(* PLC project Sin nombre, Desconocido Sin nombre 1 *)
(* stored: creationDateTime 2024-04-04T13:22:05, modificationDateTime 2024-04-09T02:45:14 *)

PROGRAM program0
  VAR
    boton_inicio AT %IX0.0 : BOOL;  (* El boton de inicio *)
    boton_parada AT %IX0.1 : BOOL;  (* El boton para detener todo *)
    sensor_caja AT %IW0 : WORD;  (* Entrada con el sensor analogo *)
    motor_cinta AT %QX0.0 : BOOL;  (* Motor para la cinta transportadora *)
    motor_rodillo AT %QX0.1 : BOOL;  (* Motor para activar el rodillo *)
  END_VAR
  VAR
    auxiliar_inicio : BOOL;  (* Variable auxiliar para almacenar si se presiono el boton de inicio *)
    auxiliar_sensor : BOOL;  (* Variable auxiliar para determinar si el sensor esta detectando la caja *)
    auxiliar_reloj : BOOL;  (* Variable auxiliar para determinar si el reloj esta contando *)
    sensor_esta_conectado : BOOL;  (* Comprobacion de que el sensor esta funcionando *)
    sensor_tapado : BOOL;  (* Comprobacion de que el sensor esta siendo tapado *)
  END_VAR
  VAR CONSTANT
    min_luz : WORD := 3500;  (* Minimo de luz requerida para saber si el sensor esta siendo tapado o no *)
    max_tiempo_rodillo : TIME := T#500ms;  (* Maxima cantidad de tiempo por la que el motor del rodillo esta activo *)
  END_VAR
  VAR
    reloj : TOF;  (* Funcion de reloj *)
  END_VAR

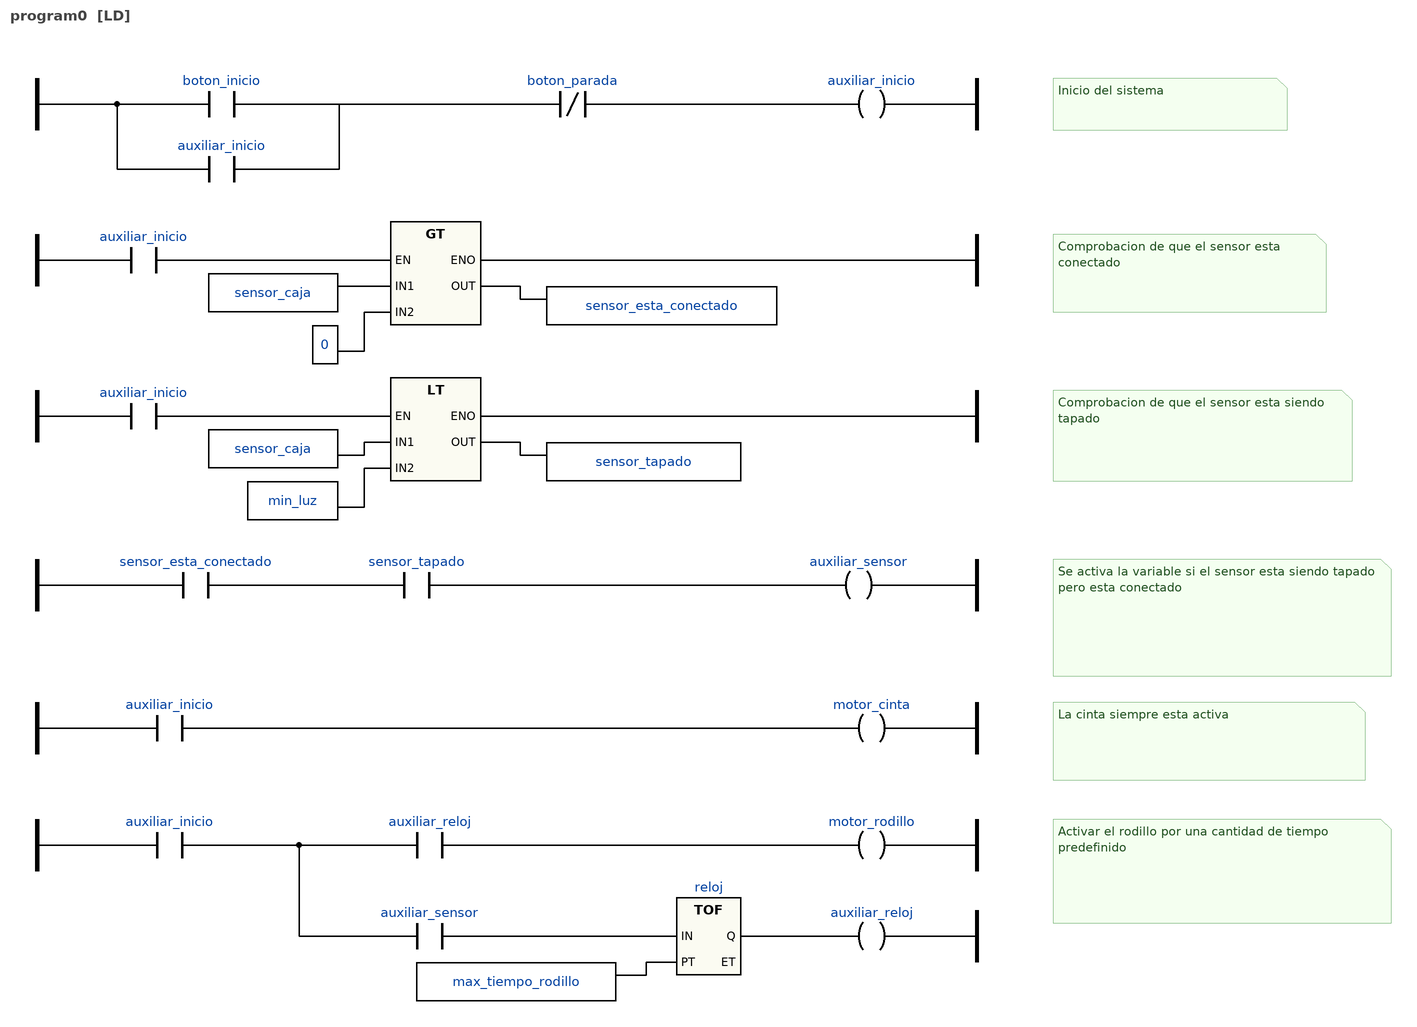
(* LD diagram, written out as Structured Text *)
(* Inicio del sistema *)
auxiliar_inicio := (boton_inicio OR auxiliar_inicio) AND NOT boton_parada;
(* Comprobacion de que el sensor esta conectado *)
(* Comprobacion de que el sensor esta siendo tapado *)
(* Se activa la variable si el sensor esta siendo tapado pero esta conectado *)
(* La cinta siempre esta activa *)
(* Activar el rodillo por una cantidad de tiempo predefinido *)
reloj(IN := auxiliar_inicio AND auxiliar_sensor, PT := max_tiempo_rodillo);
auxiliar_reloj := reloj.Q;
IF auxiliar_inicio THEN sensor_esta_conectado := sensor_caja > 0; END_IF;
IF auxiliar_inicio THEN sensor_tapado := sensor_caja < min_luz; END_IF;
auxiliar_sensor := sensor_esta_conectado AND sensor_tapado;
motor_cinta := auxiliar_inicio;
motor_rodillo := auxiliar_inicio AND auxiliar_reloj;
END_PROGRAM

CONFIGURATION Config0
  RESOURCE Res0 ON PLC
    TASK task0(INTERVAL := T#20ms, PRIORITY := 0);
    PROGRAM instance0 WITH task0 : program0;
  END_RESOURCE
END_CONFIGURATION
